# EPICS substitutions: mc05/tpmacApp/Db/autohome.substitutions
file "$(EPICS_BASE)/db/autohome.db"
{

pattern
{SYS,              DEV,                 PLC,  PORT  }
{"XF:23ID1-BI",  "{Diag:3-Ax:Y}",      8     P0    }
}
